TYPE RedundancyStatus :
STRUCT
	ENO :  BOOL; 			// Redundans är aktiverad
	UPPSTART_DONE:BOOL;
	TF_CMD:BOOL;
	TF_V:BOOL;
	TF_OP:REAL;
	TL_GP_PV:REAL;
	FF_CMD:BOOL;
	FF_V:BOOL;
	FF_OP:REAL;
	FL_GP_PV:REAL;
	SERVICEBRYTARE:BOOL;
END_STRUCT
END_TYPE

(* stored: Version 1.1.0.1, ProductVersion 3.1.4024.6
   DUT RedundancyStatus: Id {372915a6-6c25-4b90-a203-c466ec57e205} *)
